# EPICS StreamDevice protocol: Mixer.proto
##################################################
# General Settings
##################################################

Terminator = CR;
ReplyTimeout = 1000;
locktimeout = 5000;
readtimeout  = 1000;
extrainput   = Ignore;

###################################################
# Get functions
###################################################

writePosition {
   out "%i";
   in "OK";
}

#Get Mixer Position
getPosition{
   out "P";
   in "%i";
}
